// TIA Portal V17 program export: 0 tag tables, 0 data types, 0 data blocks, 2 code blocks (in call order from the OBs), 0 instance data blocks

ORGANIZATION_BLOCK "Main"   // OB1, LAD, ProgramCycle
TITLE = "Main Program Sweep (Cycle)"
{ S7_Optimized_Access := 'TRUE' }
VERSION : 0.1
// stored: AutoNumber true, IsIECCheckEnabled false, SetENOAutomatically false
   VAR_INPUT
      Initial_Call : Bool;   // Initial call of this OB
      Remanence : Bool;   // =True, if remanent data are available
   END_VAR
BEGIN

REGION Network 1
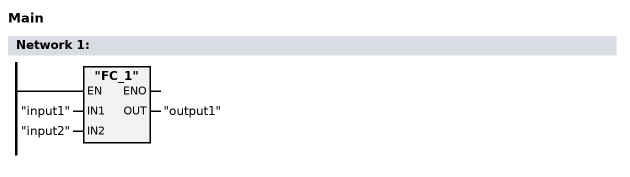
   RUNG wire#powerrail
      "FC_1"(IN1 := "input1", IN2 := "input2", OUT => "output1")
   END_RUNG
   // the same network as SCL:
   "FC_1"(IN1 := "input1", IN2 := "input2", OUT => "output1");
END_REGION
END_ORGANIZATION_BLOCK

FUNCTION "FC_1" : Void   // FC1, LAD
{ S7_Optimized_Access := 'TRUE' }
VERSION : 0.1
// stored: AutoNumber true, IsIECCheckEnabled false, SetENOAutomatically false, UDAEnableTagReadback false
   VAR_INPUT
      IN1 : Bool;
      IN2 : Bool;
   END_VAR
   VAR_OUTPUT
      OUT : Bool;
   END_VAR
BEGIN

REGION Network 1
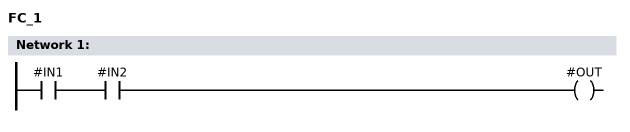
   RUNG wire#powerrail
      Contact( #IN1 )
      Contact( #IN2 )
      Coil( #OUT )
   END_RUNG
   // the same network as SCL:
   #OUT := #IN1 AND #IN2;
END_REGION
END_FUNCTION
